TYPE ST_ValveMask128 :
STRUCT
    dwLow  : DWORD;
    dwHigh : DWORD;
END_STRUCT
END_TYPE

(* stored: Version 1.1.0.1
   DUT ST_ValveMask128: Id {ee0d7dd1-9169-48a8-908f-2c505ffcb5c9} *)
